(* Logix 5000 project; controller SX_V040001_C001 vendor 1 type 14 code 77 rev 16.22; software revision 16.04; part 14 of 35 *)
(* tags used below, declared in another part *)
   ALL_KINDS : INT[90];
   DRIVE : INT[32];
   G_DInput : DINT[3];
   G_DOutput : DINT[3];
   HANDSHAKE_VISIWIN : INT[3];
   loading : INT[19];
   louvre : INT[11];
   m_alarm_exist : BOOL;
   METERING : INT[44];
   PARAMETER : INT[501];
   T_LOADING_RELEASE : TIMER;
(* MainProgram, continued *)

ROUTINE HandshakeVisiWin   (* ladder *)
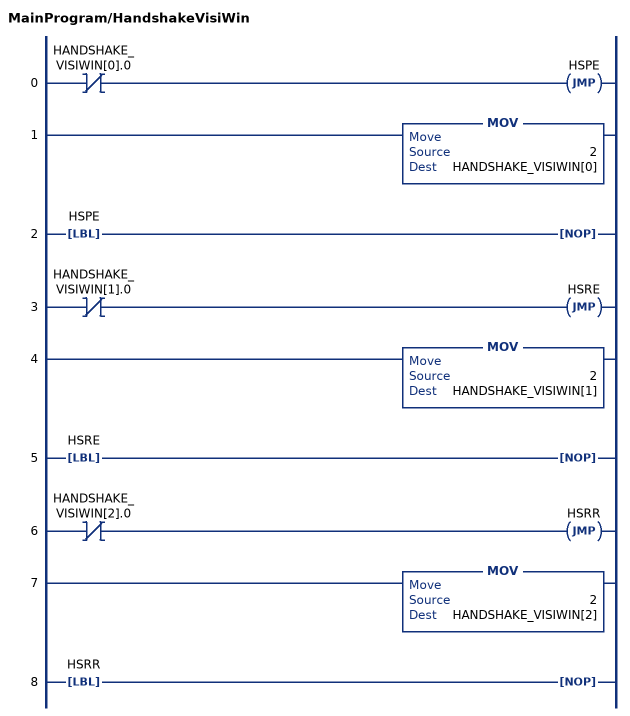
   0: XIO(HANDSHAKE_VISIWIN[0].0)JMP(HSPE);
   1: MOV(2,HANDSHAKE_VISIWIN[0]);
   2: LBL(HSPE)NOP();
   3: XIO(HANDSHAKE_VISIWIN[1].0)JMP(HSRE);
   4: MOV(2,HANDSHAKE_VISIWIN[1]);
   5: LBL(HSRE)NOP();
   6: XIO(HANDSHAKE_VISIWIN[2].0)JMP(HSRR);
   7: MOV(2,HANDSHAKE_VISIWIN[2]);
   8: LBL(HSRR)NOP();
END_ROUTINE

ROUTINE Loading   (* ladder *)
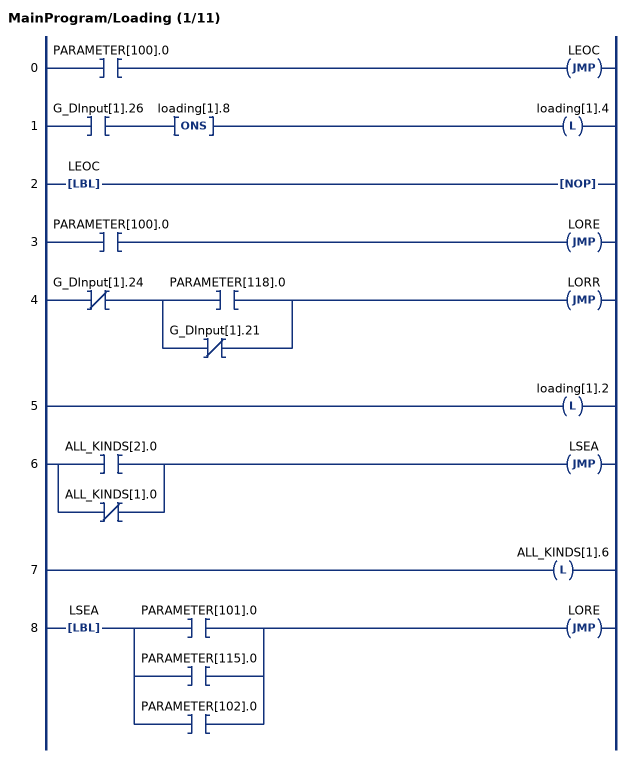
   0: XIC(PARAMETER[100].0)JMP(LEOC);
   1: XIC(G_DInput[1].26)ONS(loading[1].8)OTL(loading[1].4);
   2: LBL(LEOC)NOP();
   3: XIC(PARAMETER[100].0)JMP(LORE);
   4: XIO(G_DInput[1].24)[XIC(PARAMETER[118].0) ,XIO(G_DInput[1].21) ]JMP(LORR);
   5: OTL(loading[1].2);
   6: [XIC(ALL_KINDS[2].0) ,XIO(ALL_KINDS[1].0) ]JMP(LSEA);
   7: OTL(ALL_KINDS[1].6);
   8: LBL(LSEA)[XIC(PARAMETER[101].0) ,XIC(PARAMETER[115].0) ,XIC(PARAMETER[102].0) ]JMP(LORE);
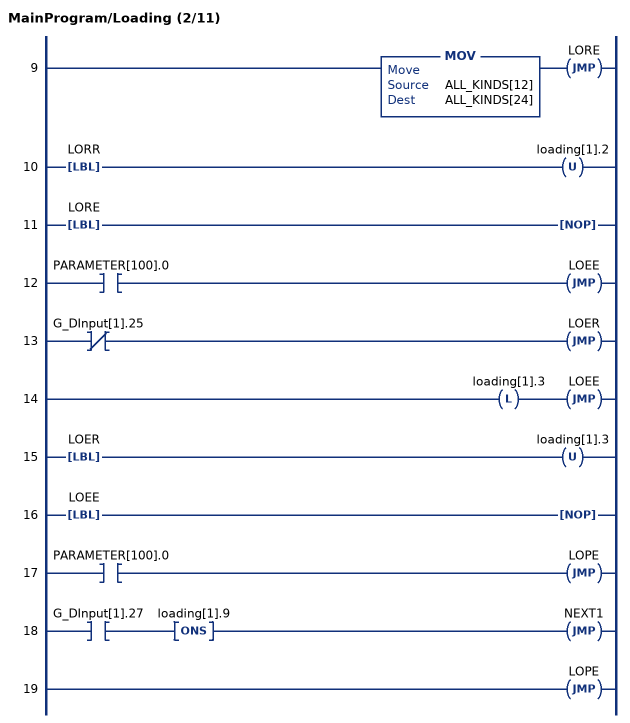
   9: MOV(ALL_KINDS[12],ALL_KINDS[24])JMP(LORE);
   10: LBL(LORR)OTU(loading[1].2);
   11: LBL(LORE)NOP();
   12: XIC(PARAMETER[100].0)JMP(LOEE);
   13: XIO(G_DInput[1].25)JMP(LOER);
   14: OTL(loading[1].3)JMP(LOEE);
   15: LBL(LOER)OTU(loading[1].3);
   16: LBL(LOEE)NOP();
   17: XIC(PARAMETER[100].0)JMP(LOPE);
   18: XIC(G_DInput[1].27)ONS(loading[1].9)JMP(NEXT1);
   19: JMP(LOPE);
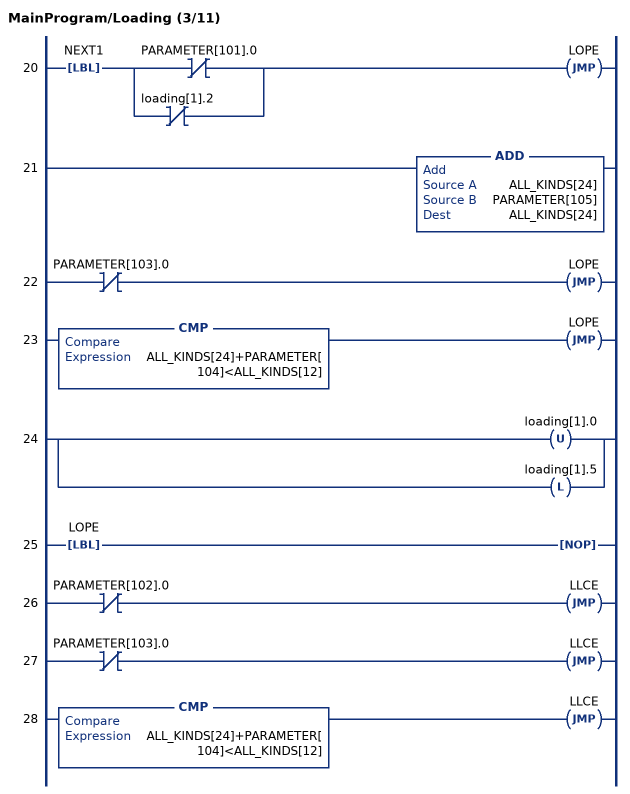
   20: LBL(NEXT1)[XIO(PARAMETER[101].0) ,XIO(loading[1].2) ]JMP(LOPE);
   21: ADD(ALL_KINDS[24],PARAMETER[105],ALL_KINDS[24]);
   22: XIO(PARAMETER[103].0)JMP(LOPE);
   23: CMP(ALL_KINDS[24]+PARAMETER[104]<ALL_KINDS[12])JMP(LOPE);
   24: [OTU(loading[1].0) ,OTL(loading[1].5) ];
   25: LBL(LOPE)NOP();
   26: XIO(PARAMETER[102].0)JMP(LLCE);
   27: XIO(PARAMETER[103].0)JMP(LLCE);
   28: CMP(ALL_KINDS[24]+PARAMETER[104]<ALL_KINDS[12])JMP(LLCE);
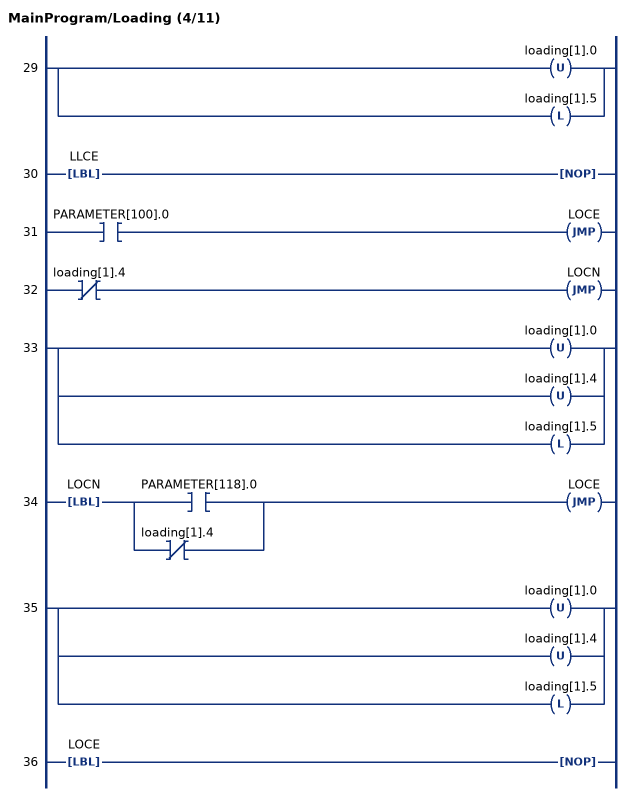
   29: [OTU(loading[1].0) ,OTL(loading[1].5) ];
   30: LBL(LLCE)NOP();
   31: XIC(PARAMETER[100].0)JMP(LOCE);
   32: XIO(loading[1].4)JMP(LOCN);
   33: [OTU(loading[1].0) ,OTU(loading[1].4) ,OTL(loading[1].5) ];
   34: LBL(LOCN)[XIC(PARAMETER[118].0) ,XIO(loading[1].4) ]JMP(LOCE);
   35: [OTU(loading[1].0) ,OTU(loading[1].4) ,OTL(loading[1].5) ];
   36: LBL(LOCE)NOP();
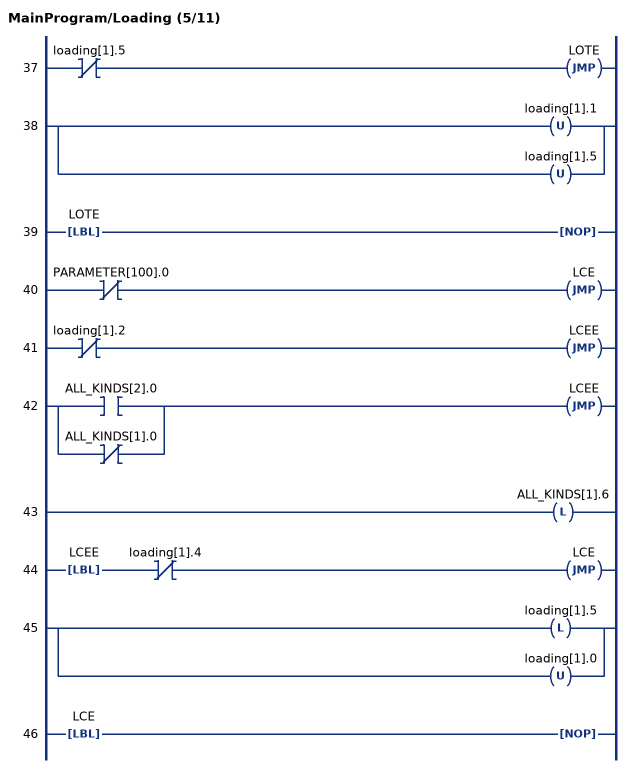
   37: XIO(loading[1].5)JMP(LOTE);
   38: [OTU(loading[1].1) ,OTU(loading[1].5) ];
   39: LBL(LOTE)NOP();
   40: XIO(PARAMETER[100].0)JMP(LCE);
   41: XIO(loading[1].2)JMP(LCEE);
   42: [XIC(ALL_KINDS[2].0) ,XIO(ALL_KINDS[1].0) ]JMP(LCEE);
   43: OTL(ALL_KINDS[1].6);
   44: LBL(LCEE)XIO(loading[1].4)JMP(LCE);
   45: [OTL(loading[1].5) ,OTU(loading[1].0) ];
   46: LBL(LCE)NOP();
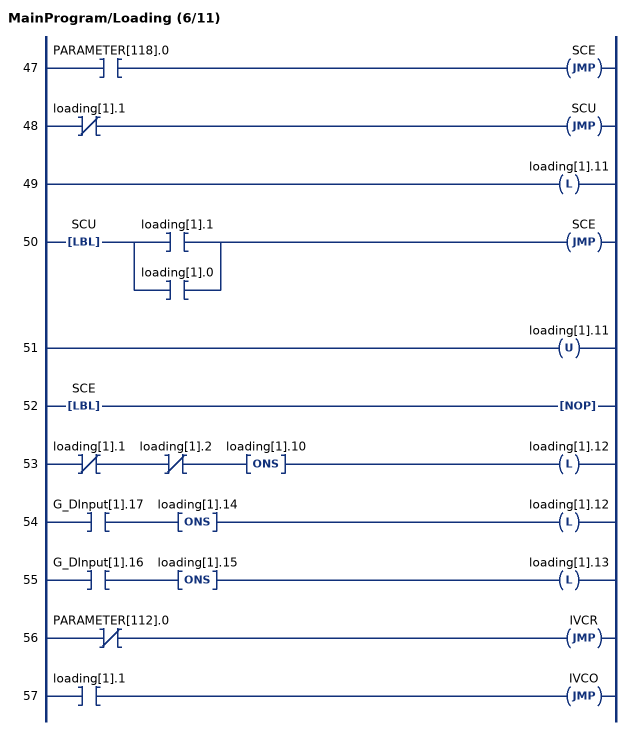
   47: XIC(PARAMETER[118].0)JMP(SCE);
   48: XIO(loading[1].1)JMP(SCU);
   49: OTL(loading[1].11);
   50: LBL(SCU)[XIC(loading[1].1) ,XIC(loading[1].0) ]JMP(SCE);
   51: OTU(loading[1].11);
   52: LBL(SCE)NOP();
   53: XIO(loading[1].1)XIO(loading[1].2)ONS(loading[1].10)OTL(loading[1].12);
   54: XIC(G_DInput[1].17)ONS(loading[1].14)OTL(loading[1].12);
   55: XIC(G_DInput[1].16)ONS(loading[1].15)OTL(loading[1].13);
   56: XIO(PARAMETER[112].0)JMP(IVCR);
   57: XIC(loading[1].1)JMP(IVCO);
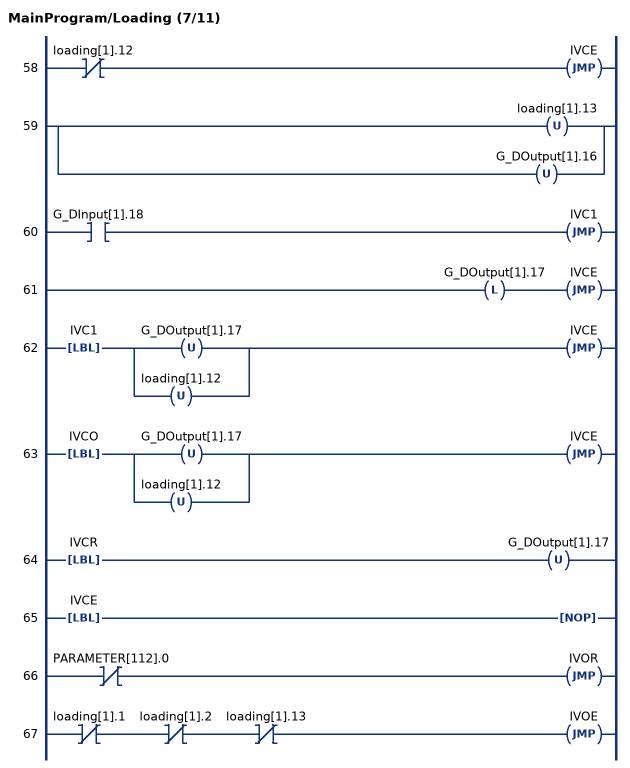
   58: XIO(loading[1].12)JMP(IVCE);
   59: [OTU(loading[1].13) ,OTU(G_DOutput[1].16) ];
   60: XIC(G_DInput[1].18)JMP(IVC1);
   61: OTL(G_DOutput[1].17)JMP(IVCE);
   62: LBL(IVC1)[OTU(G_DOutput[1].17) ,OTU(loading[1].12) ]JMP(IVCE);
   63: LBL(IVCO)[OTU(G_DOutput[1].17) ,OTU(loading[1].12) ]JMP(IVCE);
   64: LBL(IVCR)OTU(G_DOutput[1].17);
   65: LBL(IVCE)NOP();
   66: XIO(PARAMETER[112].0)JMP(IVOR);
   67: XIO(loading[1].1)XIO(loading[1].2)XIO(loading[1].13)JMP(IVOE);
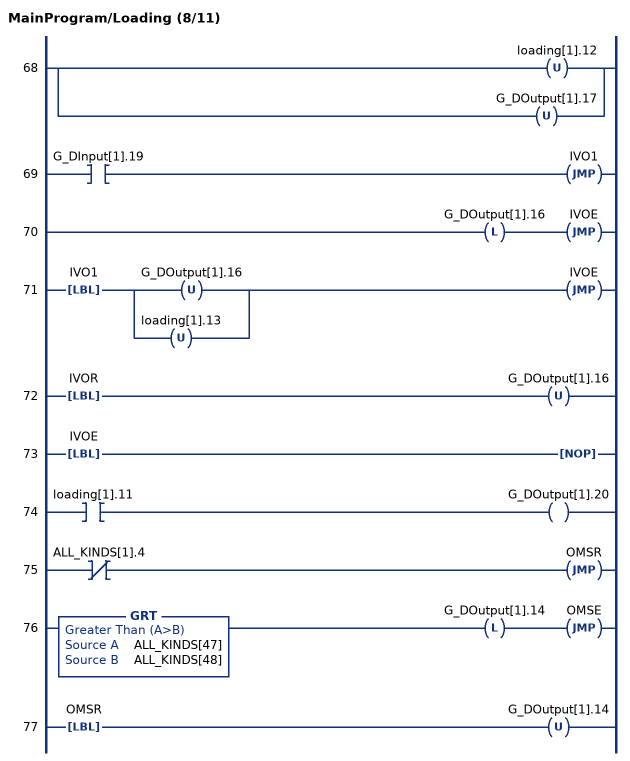
   68: [OTU(loading[1].12) ,OTU(G_DOutput[1].17) ];
   69: XIC(G_DInput[1].19)JMP(IVO1);
   70: OTL(G_DOutput[1].16)JMP(IVOE);
   71: LBL(IVO1)[OTU(G_DOutput[1].16) ,OTU(loading[1].13) ]JMP(IVOE);
   72: LBL(IVOR)OTU(G_DOutput[1].16);
   73: LBL(IVOE)NOP();
   74: XIC(loading[1].11)OTE(G_DOutput[1].20);
   75: XIO(ALL_KINDS[1].4)JMP(OMSR);
   76: GRT(ALL_KINDS[47],ALL_KINDS[48])OTL(G_DOutput[1].14)JMP(OMSE);
   77: LBL(OMSR)OTU(G_DOutput[1].14);
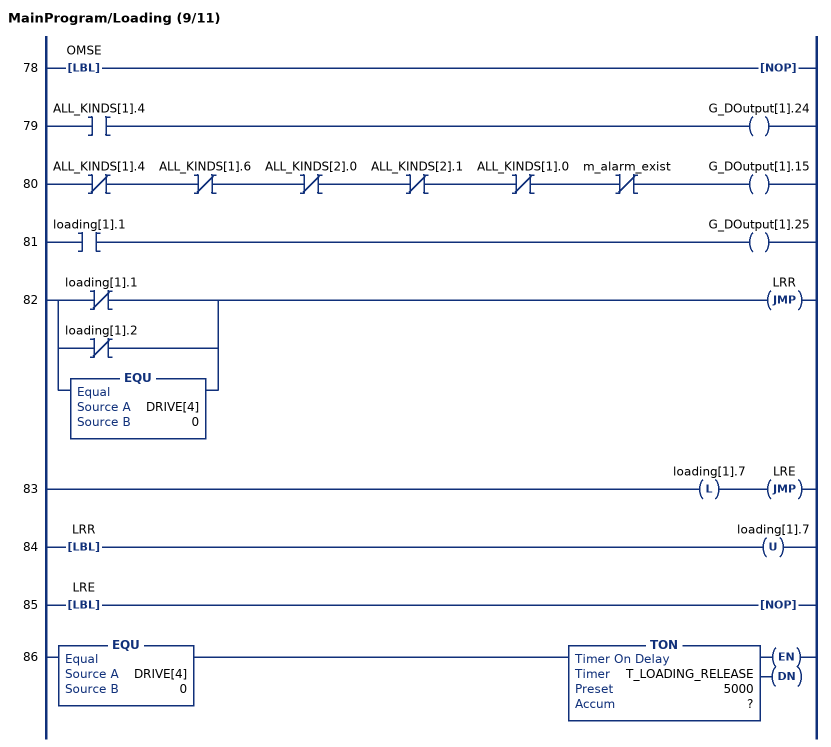
   78: LBL(OMSE)NOP();
   79: XIC(ALL_KINDS[1].4)OTE(G_DOutput[1].24);
   80: XIO(ALL_KINDS[1].4)XIO(ALL_KINDS[1].6)XIO(ALL_KINDS[2].0)XIO(ALL_KINDS[2].1)XIO(ALL_KINDS[1].0)XIO(m_alarm_exist)OTE(G_DOutput[1].15);
   81: XIC(loading[1].1)OTE(G_DOutput[1].25);
   82: [XIO(loading[1].1) ,XIO(loading[1].2) ,EQU(DRIVE[4],0) ]JMP(LRR);
   83: OTL(loading[1].7)JMP(LRE);
   84: LBL(LRR)OTU(loading[1].7);
   85: LBL(LRE)NOP();
   86: EQU(DRIVE[4],0)TON(T_LOADING_RELEASE,?,?);
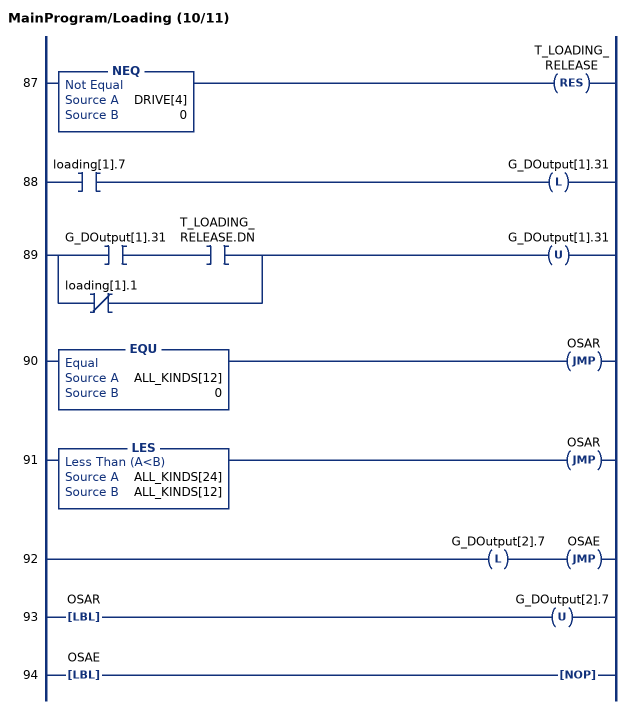
   87: NEQ(DRIVE[4],0)RES(T_LOADING_RELEASE);
   88: XIC(loading[1].7)OTL(G_DOutput[1].31);
   89: [XIC(G_DOutput[1].31) XIC(T_LOADING_RELEASE.DN) ,XIO(loading[1].1) ]OTU(G_DOutput[1].31);
   90: EQU(ALL_KINDS[12],0)JMP(OSAR);
   91: LES(ALL_KINDS[24],ALL_KINDS[12])JMP(OSAR);
   92: OTL(G_DOutput[2].7)JMP(OSAE);
   93: LBL(OSAR)OTU(G_DOutput[2].7);
   94: LBL(OSAE)NOP();
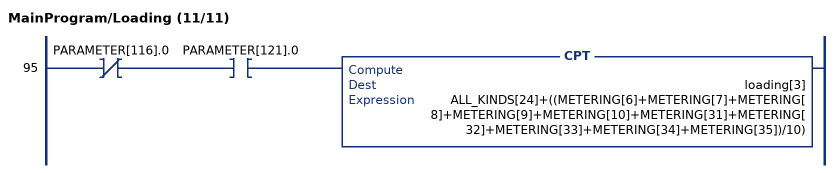
   95: XIO(PARAMETER[116].0)XIC(PARAMETER[121].0)CPT(loading[3],ALL_KINDS[24]+((METERING[6]+METERING[7]+METERING[8]+METERING[9]+METERING[10]+METERING[31]+METERING[32]+METERING[33]+METERING[34]+METERING[35])/10));
END_ROUTINE

ROUTINE Louvre23Pneum   (* ladder *)
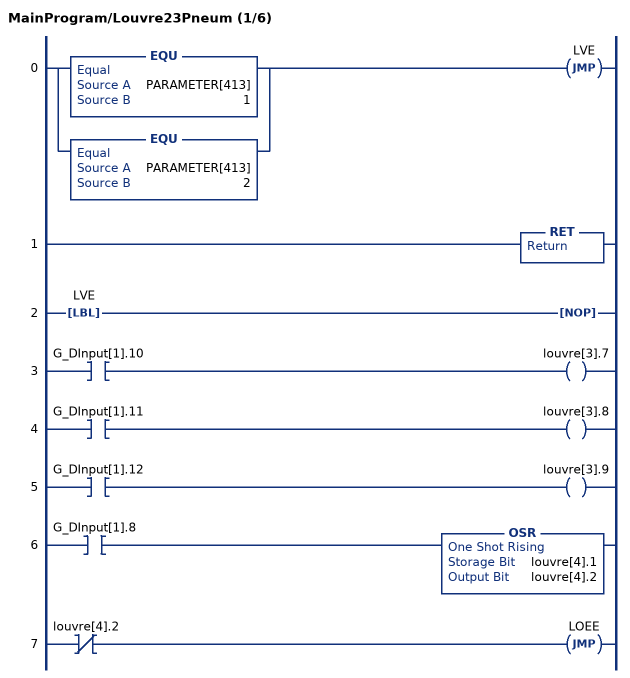
   0: [EQU(PARAMETER[413],1) ,EQU(PARAMETER[413],2) ]JMP(LVE);
   1: RET();
   2: LBL(LVE)NOP();
   3: XIC(G_DInput[1].10)OTE(louvre[3].7);
   4: XIC(G_DInput[1].11)OTE(louvre[3].8);
   5: XIC(G_DInput[1].12)OTE(louvre[3].9);
   6: XIC(G_DInput[1].8)OSR(louvre[4].1,louvre[4].2);
   7: XIO(louvre[4].2)JMP(LOEE);
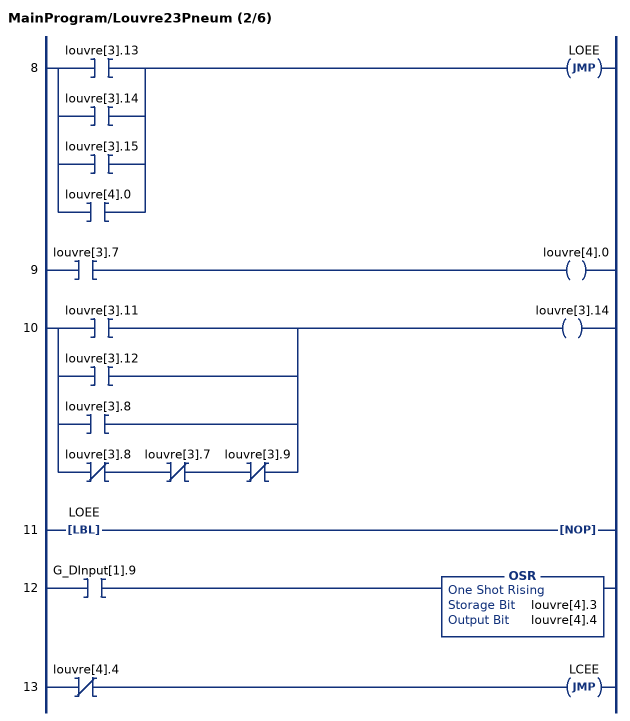
   8: [XIC(louvre[3].13) ,XIC(louvre[3].14) ,XIC(louvre[3].15) ,XIC(louvre[4].0) ]JMP(LOEE);
   9: XIC(louvre[3].7)OTE(louvre[4].0);
   10: [XIC(louvre[3].11) ,XIC(louvre[3].12) ,XIC(louvre[3].8) ,XIO(louvre[3].8) XIO(louvre[3].7) XIO(louvre[3].9) ]OTE(louvre[3].14);
   11: LBL(LOEE)NOP();
   12: XIC(G_DInput[1].9)OSR(louvre[4].3,louvre[4].4);
   13: XIO(louvre[4].4)JMP(LCEE);
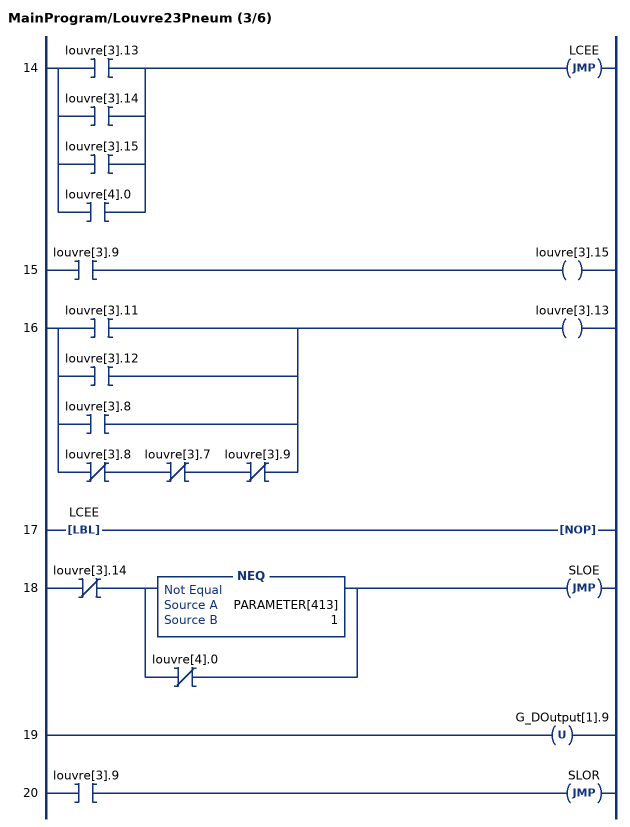
   14: [XIC(louvre[3].13) ,XIC(louvre[3].14) ,XIC(louvre[3].15) ,XIC(louvre[4].0) ]JMP(LCEE);
   15: XIC(louvre[3].9)OTE(louvre[3].15);
   16: [XIC(louvre[3].11) ,XIC(louvre[3].12) ,XIC(louvre[3].8) ,XIO(louvre[3].8) XIO(louvre[3].7) XIO(louvre[3].9) ]OTE(louvre[3].13);
   17: LBL(LCEE)NOP();
   18: XIO(louvre[3].14)[NEQ(PARAMETER[413],1) ,XIO(louvre[4].0) ]JMP(SLOE);
   19: OTU(G_DOutput[1].9);
   20: XIC(louvre[3].9)JMP(SLOR);
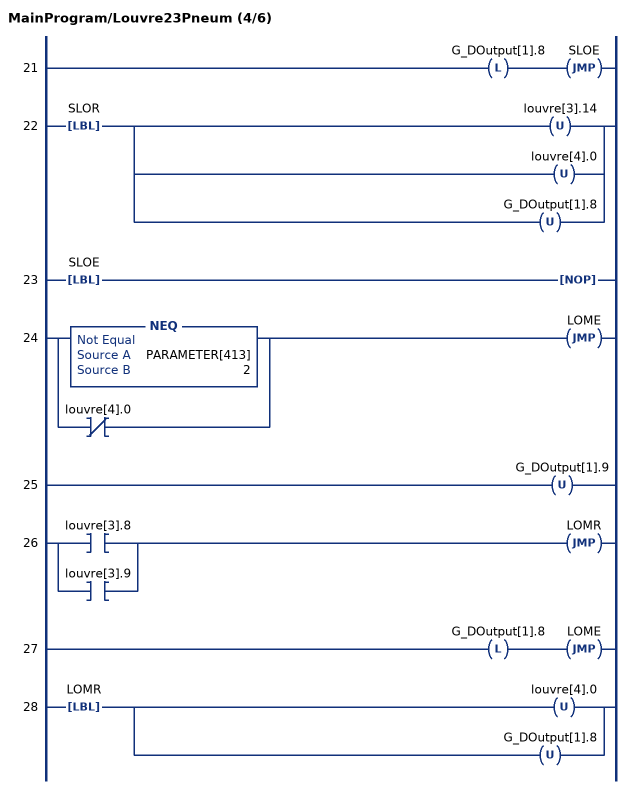
   21: OTL(G_DOutput[1].8)JMP(SLOE);
   22: LBL(SLOR)[OTU(louvre[3].14) ,OTU(louvre[4].0) ,OTU(G_DOutput[1].8) ];
   23: LBL(SLOE)NOP();
   24: [NEQ(PARAMETER[413],2) ,XIO(louvre[4].0) ]JMP(LOME);
   25: OTU(G_DOutput[1].9);
   26: [XIC(louvre[3].8) ,XIC(louvre[3].9) ]JMP(LOMR);
   27: OTL(G_DOutput[1].8)JMP(LOME);
   28: LBL(LOMR)[OTU(louvre[4].0) ,OTU(G_DOutput[1].8) ];
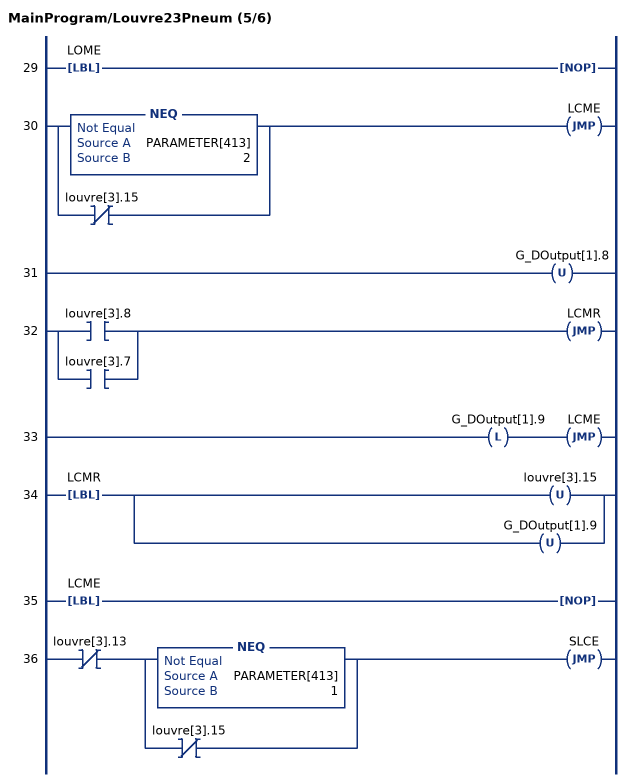
   29: LBL(LOME)NOP();
   30: [NEQ(PARAMETER[413],2) ,XIO(louvre[3].15) ]JMP(LCME);
   31: OTU(G_DOutput[1].8);
   32: [XIC(louvre[3].8) ,XIC(louvre[3].7) ]JMP(LCMR);
   33: OTL(G_DOutput[1].9)JMP(LCME);
   34: LBL(LCMR)[OTU(louvre[3].15) ,OTU(G_DOutput[1].9) ];
   35: LBL(LCME)NOP();
   36: XIO(louvre[3].13)[NEQ(PARAMETER[413],1) ,XIO(louvre[3].15) ]JMP(SLCE);
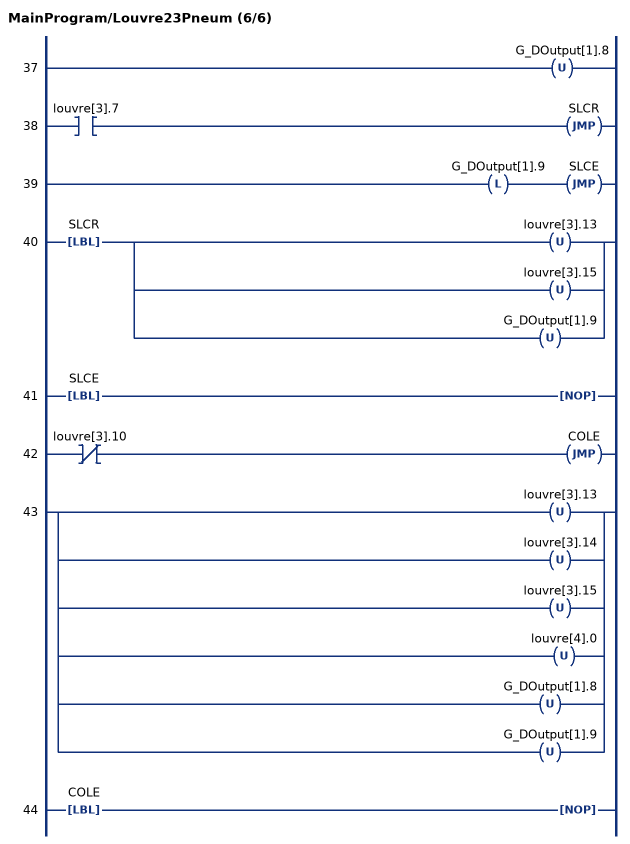
   37: OTU(G_DOutput[1].8);
   38: XIC(louvre[3].7)JMP(SLCR);
   39: OTL(G_DOutput[1].9)JMP(SLCE);
   40: LBL(SLCR)[OTU(louvre[3].13) ,OTU(louvre[3].15) ,OTU(G_DOutput[1].9) ];
   41: LBL(SLCE)NOP();
   42: XIO(louvre[3].10)JMP(COLE);
   43: [OTU(louvre[3].13) ,OTU(louvre[3].14) ,OTU(louvre[3].15) ,OTU(louvre[4].0) ,OTU(G_DOutput[1].8) ,OTU(G_DOutput[1].9) ];
   44: LBL(COLE)NOP();
END_ROUTINE
